{attribute 'GeneratedUsingTerminal: EL5151-0021-0018'}
{attribute addProperty BoxType "EL5151-0021-0018"}
{attribute addProperty Id "StatusAT %I*Status_3BE3BF2611Counter_valueAT %I*UDINT4Latch_valueAT %I*UDINT4"}
{attribute addProperty CRC "2891038912"}
{attribute addProperty Size "19"}
TYPE ENC_Status_AC51C0C0 EXTENDS InputBase_8311D824 :
STRUCT
	{attribute addProperty Name "Status"}
	Status AT %I* : Status_3BE3BF26;
	{attribute addProperty Name "Counter_value"}
	Counter_value AT %I* : UDINT;
	{attribute addProperty Name "Latch_value"}
	Latch_value AT %I* : UDINT;
END_STRUCT
END_TYPE

(* stored: Version 1.2.0.0, ProductVersion 3.1.4024.9
   DUT ENC_Status_AC51C0C0: Id {aac5afc1-274b-485d-bb37-3d7837b842a2} *)
